DATA_BLOCK "teste_DB"
{ S7_Optimized_Access := 'TRUE' }
VERSION : 0.1
NON_RETAIN
"teste"

BEGIN

END_DATA_BLOCK

